// TIA Portal V17 export
// export: Created 2025-06-26T06:49:11.8212921Z, ExportSetting WithDefaults, DisplayName Totally Integrated Automation Portal, DisplayVersion V17 Update 8, DisplayName TIA Portal Openness, DisplayVersion V17 Update 8, DisplayName TIA Portal Version Control Interface, DisplayVersion V17, DisplayName STEP 7 Professional, DisplayVersion V17 Update 8, DisplayName STEP 7 Safety, DisplayVersion V17 Update 6, DisplayName WinCC Advanced, DisplayVersion V17 Update 8
FUNCTION_BLOCK "Regulation"   // FB5, FBD
{ S7_Optimized_Access := 'TRUE' }
VERSION : 0.1
// stored: AutoNumber true, IsIECCheckEnabled true, IsRetainMemResEnabled false, MemoryReserve 10, SetENOAutomatically false, UDAEnableTagReadback false
   VAR
      ExpValveCurrentPressureLimitation : Bool;
      enEmergencyStop { ExternalAccessible := 'False'; ExternalVisible := 'False'; ExternalWritable := 'False'} : Bool;
      CPCPumpRequestFromCPC { ExternalAccessible := 'False'; ExternalVisible := 'False'; ExternalWritable := 'False'} : Bool;   // Crankcase Pressure Control wants to run CPC pump
      CPCPumpRequestFromPurge { ExternalAccessible := 'False'; ExternalVisible := 'False'; ExternalWritable := 'False'} : Bool;   // Do compressor manifold purge
      ExpValveCurrentPressureTarged : Real;
      PerformanceControl_PerformanceRate : Real;
      PerformanceControl { ExternalAccessible := 'False'; ExternalVisible := 'False'; ExternalWritable := 'False'; S7_SetPoint := 'True'} : "PerformanceControl";   // Compressor setpoint
      SuperheatControl { ExternalAccessible := 'False'; ExternalVisible := 'False'; ExternalWritable := 'False'; S7_SetPoint := 'True'} : "SuperheatControl";   // Superheat setpoint
      PinchControl { ExternalAccessible := 'False'; ExternalVisible := 'False'; ExternalWritable := 'False'; S7_SetPoint := 'True'} : "PinchControl";
      CrankcaseOilHeating { ExternalAccessible := 'False'; ExternalVisible := 'False'; ExternalWritable := 'False'; S7_SetPoint := 'True'} : "OilHeating";
      MotorSpeedControl { ExternalAccessible := 'False'; ExternalVisible := 'False'; ExternalWritable := 'False'; S7_SetPoint := 'True'} : "MotorControl";
      SafetyRelay { ExternalAccessible := 'False'; ExternalVisible := 'False'; ExternalWritable := 'False'; S7_SetPoint := 'True'} : "fbSafetyRelay";
      CabinetTemperature { ExternalAccessible := 'False'; ExternalVisible := 'False'; ExternalWritable := 'False'; S7_SetPoint := 'True'} : "fbTemperatureController2";
      ContainerVentilation { ExternalAccessible := 'False'; ExternalVisible := 'False'; ExternalWritable := 'False'; S7_SetPoint := 'True'} : "fbPI_Regulator";
      CrankcasePressureControl { ExternalAccessible := 'False'; ExternalVisible := 'False'; ExternalWritable := 'False'; S7_SetPoint := 'True'} : "CrankcasePressureControl";
      OilSeparator { ExternalAccessible := 'False'; ExternalVisible := 'False'; ExternalWritable := 'False'; S7_SetPoint := 'True'} : "OilSeparator";
      ShaftSealCartridge { ExternalAccessible := 'False'; ExternalVisible := 'False'; ExternalWritable := 'False'; S7_SetPoint := 'True'} : "ShaftSealCartridge";
      LubricationPriming { ExternalAccessible := 'False'; ExternalVisible := 'False'; ExternalWritable := 'False'; S7_SetPoint := 'True'} : "LubricationPriming";
      ValveControl { ExternalAccessible := 'False'; ExternalVisible := 'False'; ExternalWritable := 'False'; S7_SetPoint := 'True'} : "ValveControl";
      PurgeControl { ExternalAccessible := 'False'; ExternalVisible := 'False'; ExternalWritable := 'False'; S7_SetPoint := 'True'} : "fbPurgeControl";
      FilterDryer { S7_SetPoint := 'True'} : "fbFilterDryer";
      OilRecovery { S7_SetPoint := 'True'} : "fbOilRecovery";
      RecuperatorBypass { S7_SetPoint := 'True'} : "fbNullRegulator";
      HeatSourceCycle { S7_SetPoint := 'True'} : "fbTrackingRegulator";
      HeatSourceCyclePIP { S7_SetPoint := 'True'} : "fbPIP_Regulator";
      HeatboosterSetpointPrev { ExternalAccessible := 'False'; ExternalVisible := 'False'; ExternalWritable := 'False'} : Real;   // TEST
      HeatSinkSetpointPrev { ExternalAccessible := 'False'; ExternalVisible := 'False'; ExternalWritable := 'False'} : Real;   // TEST
      HeatSourceSetpointPrev { ExternalAccessible := 'False'; ExternalVisible := 'False'; ExternalWritable := 'False'} : Real;   // TEST
      VariableSetpointPrev { ExternalAccessible := 'False'; ExternalVisible := 'False'; ExternalWritable := 'False'} : Real;
      RegulationTarget { ExternalAccessible := 'False'; ExternalVisible := 'False'; ExternalWritable := 'False'} : Int;   // TEST
      epHeatSinkControlActive { ExternalAccessible := 'False'; ExternalVisible := 'False'; ExternalWritable := 'False'} : Bool;
      epHeatSourceControlActive { ExternalAccessible := 'False'; ExternalVisible := 'False'; ExternalWritable := 'False'} : Bool;
      epVariableControlActive { ExternalAccessible := 'False'; ExternalVisible := 'False'; ExternalWritable := 'False'} : Bool;
      TEST1 : Bool;
   END_VAR
   VAR_TEMP
      AdditionalSuperHeat : Real;
      PerformanceSetpoint : Real;
      AdditionalSuperheatPinch : Real;
   END_VAR
   VAR_TEMP   // added for the SCL form of the ladder/FBD networks
      _w1 : Bool;
   END_VAR
BEGIN

REGION Network 1: Performance control
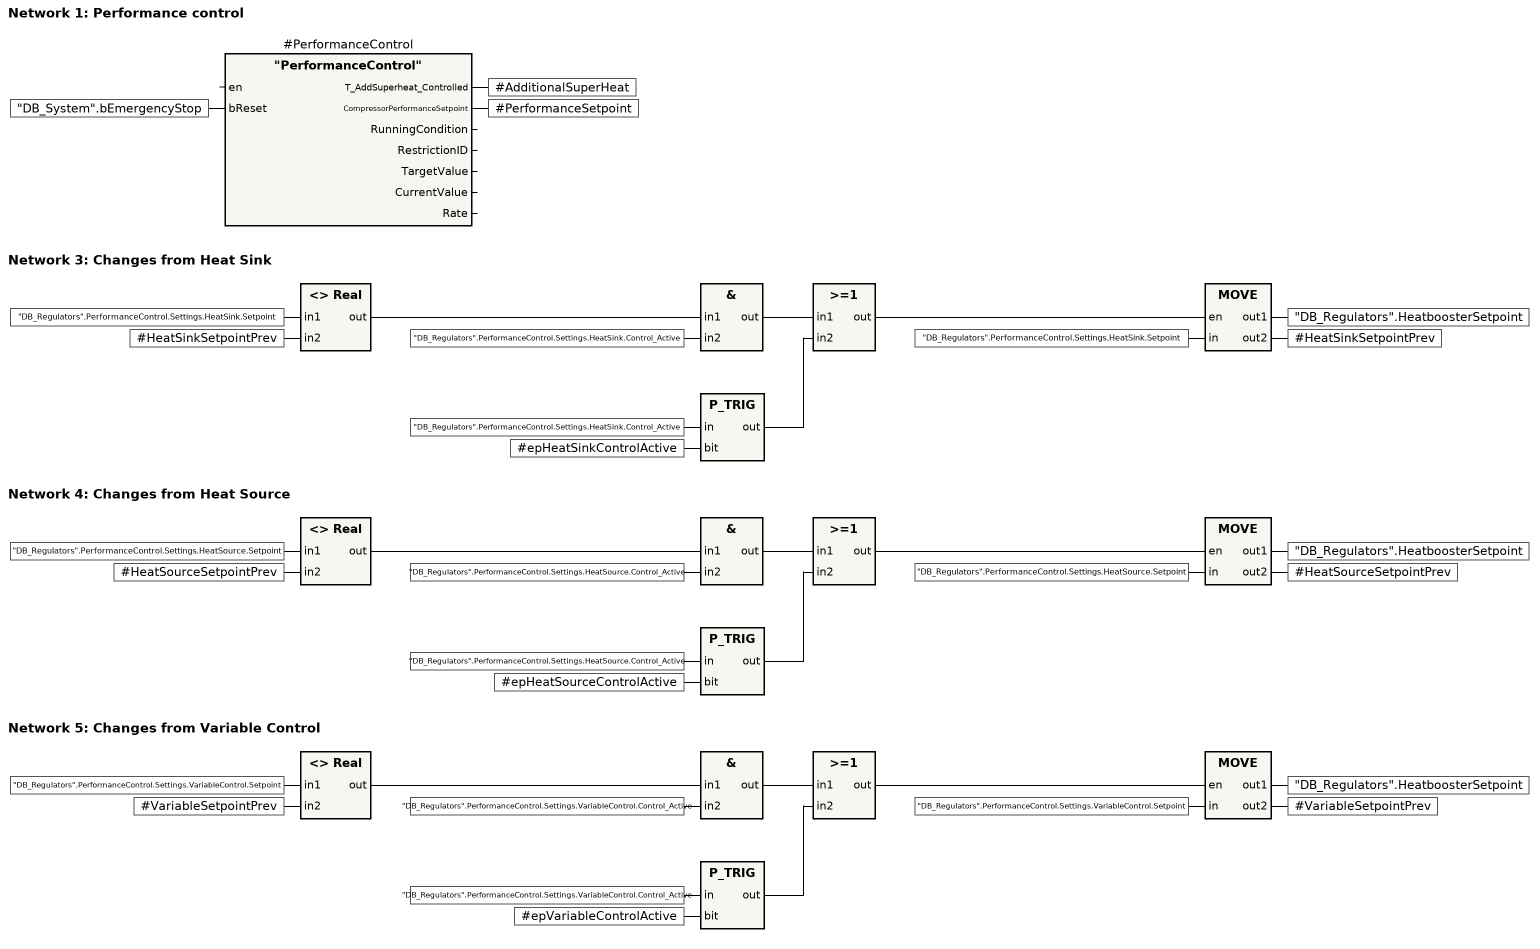
   #PerformanceControl(bReset := "DB_System".bEmergencyStop,   // "PerformanceControl"
                       T_AddSuperheat_Controlled => #AdditionalSuperHeat,
                       CompressorPerformanceSetpoint => #PerformanceSetpoint);
END_REGION

REGION Network 2 (SCL): Performance rate
   // Used in HMI only
   IF "DB_State".State."5_Warmup" OR "DB_State".State."6_Running" AND #PerformanceControl.RunningCondition = TRUE THEN
       #PerformanceControl_PerformanceRate := #MotorSpeedControl.NEngineSetpoint / 15 - #AdditionalSuperHeat / 50 * 30;
   ELSE
       #PerformanceControl_PerformanceRate := 0;
   END_IF;
END_REGION

REGION Network 3: Changes from Heat Sink
   // Propagate setpoint when controller is first activated, or if active and setpoint is changed
   #_w1 := "DB_Regulators".PerformanceControl.Settings.HeatSink.Control_Active AND NOT #epHeatSinkControlActive;   // rising edge
   #epHeatSinkControlActive := "DB_Regulators".PerformanceControl.Settings.HeatSink.Control_Active;
   IF (("DB_Regulators".PerformanceControl.Settings.HeatSink.Setpoint <> #HeatSinkSetpointPrev) AND "DB_Regulators".PerformanceControl.Settings.HeatSink.Control_Active) OR #_w1 THEN
       "DB_Regulators".HeatboosterSetpoint := "DB_Regulators".PerformanceControl.Settings.HeatSink.Setpoint;
       #HeatSinkSetpointPrev := "DB_Regulators".PerformanceControl.Settings.HeatSink.Setpoint;
   END_IF;
END_REGION

REGION Network 4: Changes from Heat Source
   // Propagate setpoint when controller is first activated, or if active and setpoint is changed
   #_w1 := "DB_Regulators".PerformanceControl.Settings.HeatSource.Control_Active AND NOT #epHeatSourceControlActive;   // rising edge
   #epHeatSourceControlActive := "DB_Regulators".PerformanceControl.Settings.HeatSource.Control_Active;
   IF (("DB_Regulators".PerformanceControl.Settings.HeatSource.Setpoint <> #HeatSourceSetpointPrev) AND "DB_Regulators".PerformanceControl.Settings.HeatSource.Control_Active) OR #_w1 THEN
       "DB_Regulators".HeatboosterSetpoint := "DB_Regulators".PerformanceControl.Settings.HeatSource.Setpoint;
       #HeatSourceSetpointPrev := "DB_Regulators".PerformanceControl.Settings.HeatSource.Setpoint;
   END_IF;
END_REGION

REGION Network 5: Changes from Variable Control
   // Propagate setpoint when controller is first activated, or if active and setpoint is changed
   #_w1 := "DB_Regulators".PerformanceControl.Settings.VariableControl.Control_Active AND NOT #epVariableControlActive;   // rising edge
   #epVariableControlActive := "DB_Regulators".PerformanceControl.Settings.VariableControl.Control_Active;
   IF (("DB_Regulators".PerformanceControl.Settings.VariableControl.Setpoint <> #VariableSetpointPrev) AND "DB_Regulators".PerformanceControl.Settings.VariableControl.Control_Active) OR #_w1 THEN
       "DB_Regulators".HeatboosterSetpoint := "DB_Regulators".PerformanceControl.Settings.VariableControl.Setpoint;
       #VariableSetpointPrev := "DB_Regulators".PerformanceControl.Settings.VariableControl.Setpoint;
   END_IF;
END_REGION

REGION Network 6 (SCL): Regulation target
   // No, I didn't suddenly develop a brain hemorrage, this mess here is on purpose:
   // 1. It is a sequence of separate IFs as it mirrors the logic in PerformanceControl
   // 2. It is tempting to re-use Restriction ID, but this can take on values other than the ones here, which we want to avoid. So the value has to be reconstructed.
   // Figure out which target is active
   "DB_Regulators".RegulationTarget := 0;  // in case none of the regulators are active, none of the IFs fire...
   IF "DB_Regulators".PerformanceControl.Settings.HeatSink.Control_Active THEN
       IF "DB_Regulators".PerformanceControl.Settings.HeatSink.UseFeedFlow THEN
           "DB_Regulators".RegulationTarget := 2;
       ELSE
           "DB_Regulators".RegulationTarget := 1;
       END_IF;
   END_IF;

   IF "DB_Regulators".PerformanceControl.Settings.HeatSource.Control_Active THEN
       IF "DB_Regulators".PerformanceControl.Settings.HeatSource.UseFeedFlow THEN
           "DB_Regulators".RegulationTarget := 4;
       ELSE
           "DB_Regulators".RegulationTarget := 3;
       END_IF;
   END_IF;

   IF "DB_Regulators".PerformanceControl.Settings.VariableControl.Control_Active AND "DB_Regulators".PerformanceControl.Settings.VariableControl.ReferenceID > 0 THEN
       "DB_Regulators".RegulationTarget := 6;
   END_IF;
END_REGION

REGION Network 7: Changes from DB_Regulators
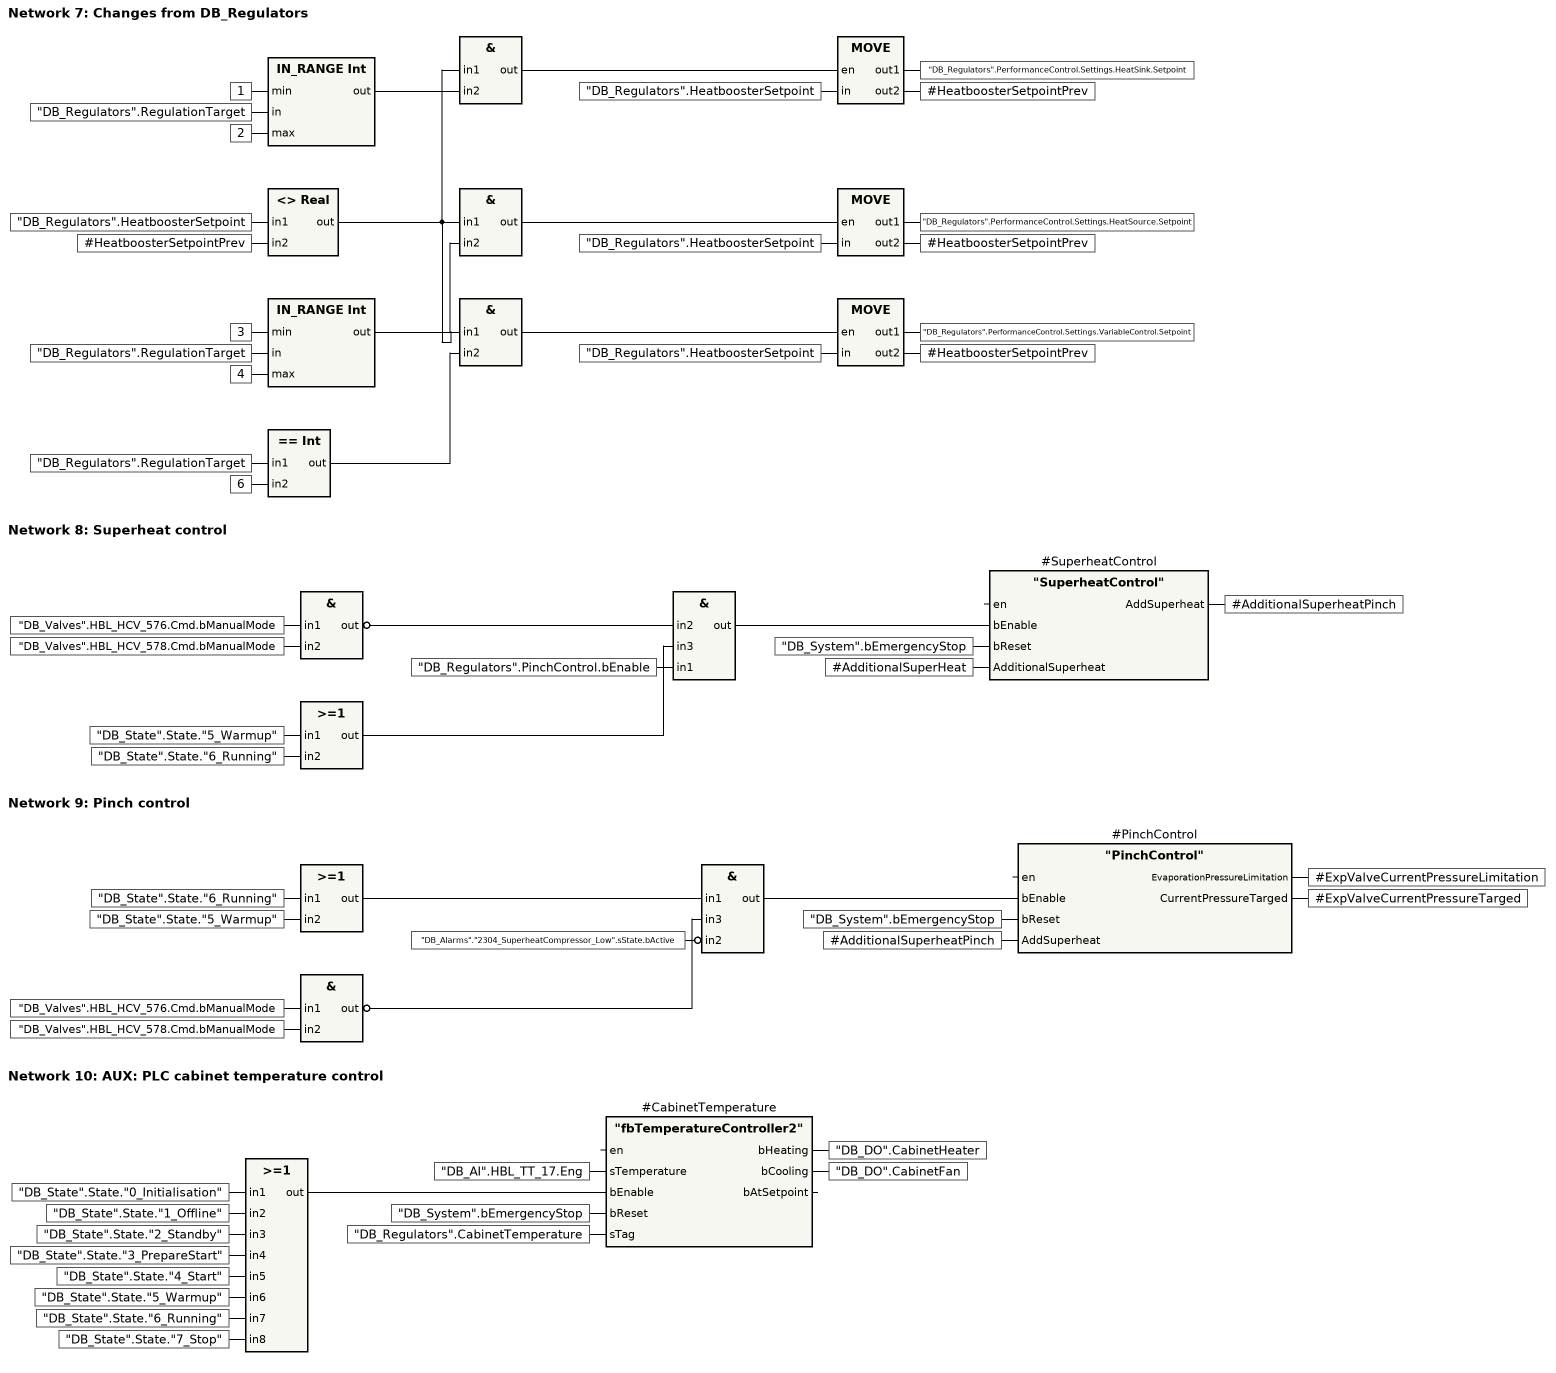
   #_w1 := "DB_Regulators".HeatboosterSetpoint <> #HeatboosterSetpointPrev;
   IF #_w1 AND (1 <= "DB_Regulators".RegulationTarget) AND ("DB_Regulators".RegulationTarget <= 2) THEN
       "DB_Regulators".PerformanceControl.Settings.HeatSink.Setpoint := "DB_Regulators".HeatboosterSetpoint;
       #HeatboosterSetpointPrev := "DB_Regulators".HeatboosterSetpoint;
   END_IF;
   IF #_w1 AND (3 <= "DB_Regulators".RegulationTarget) AND ("DB_Regulators".RegulationTarget <= 4) THEN
       "DB_Regulators".PerformanceControl.Settings.HeatSource.Setpoint := "DB_Regulators".HeatboosterSetpoint;
       #HeatboosterSetpointPrev := "DB_Regulators".HeatboosterSetpoint;
   END_IF;
   IF #_w1 AND ("DB_Regulators".RegulationTarget = 6) THEN
       "DB_Regulators".PerformanceControl.Settings.VariableControl.Setpoint := "DB_Regulators".HeatboosterSetpoint;
       #HeatboosterSetpointPrev := "DB_Regulators".HeatboosterSetpoint;
   END_IF;
END_REGION

REGION Network 8: Superheat control
   #SuperheatControl(bEnable := NOT ("DB_Valves".HBL_HCV_576.Cmd.bManualMode AND "DB_Valves".HBL_HCV_578.Cmd.bManualMode) AND ("DB_State".State."5_Warmup" OR "DB_State".State."6_Running") AND "DB_Regulators".PinchControl.bEnable,   // "SuperheatControl"
                     bReset := "DB_System".bEmergencyStop,
                     AdditionalSuperheat := #AdditionalSuperHeat,
                     AddSuperheat => #AdditionalSuperheatPinch);
END_REGION

REGION Network 9: Pinch control
   #PinchControl(bEnable := ("DB_State".State."6_Running" OR "DB_State".State."5_Warmup") AND NOT ("DB_Valves".HBL_HCV_576.Cmd.bManualMode AND "DB_Valves".HBL_HCV_578.Cmd.bManualMode) AND NOT "DB_Alarms"."2304_SuperheatCompressor_Low".sState.bActive,   // "PinchControl"
                 bReset := "DB_System".bEmergencyStop,
                 AddSuperheat := #AdditionalSuperheatPinch,
                 EvaporationPressureLimitation => #ExpValveCurrentPressureLimitation,
                 CurrentPressureTarged => #ExpValveCurrentPressureTarged);
END_REGION

REGION Network 10: AUX: PLC cabinet temperature control
   // Runs all the time, as the cabinet is running all the time...
   #CabinetTemperature(sTemperature := "DB_AI".HBL_TT_17.Eng,   // "fbTemperatureController2"
                       bEnable := "DB_State".State."0_Initialisation" OR "DB_State".State."1_Offline" OR "DB_State".State."2_Standby" OR "DB_State".State."3_PrepareStart" OR "DB_State".State."4_Start" OR "DB_State".State."5_Warmup" OR "DB_State".State."6_Running" OR "DB_State".State."7_Stop",
                       bReset := "DB_System".bEmergencyStop,
                       sTag := "DB_Regulators".CabinetTemperature,
                       bHeating => "DB_DO".CabinetHeater,
                       bCooling => "DB_DO".CabinetFan);
END_REGION

REGION Network 11: AUX: Crankcase oil heater control
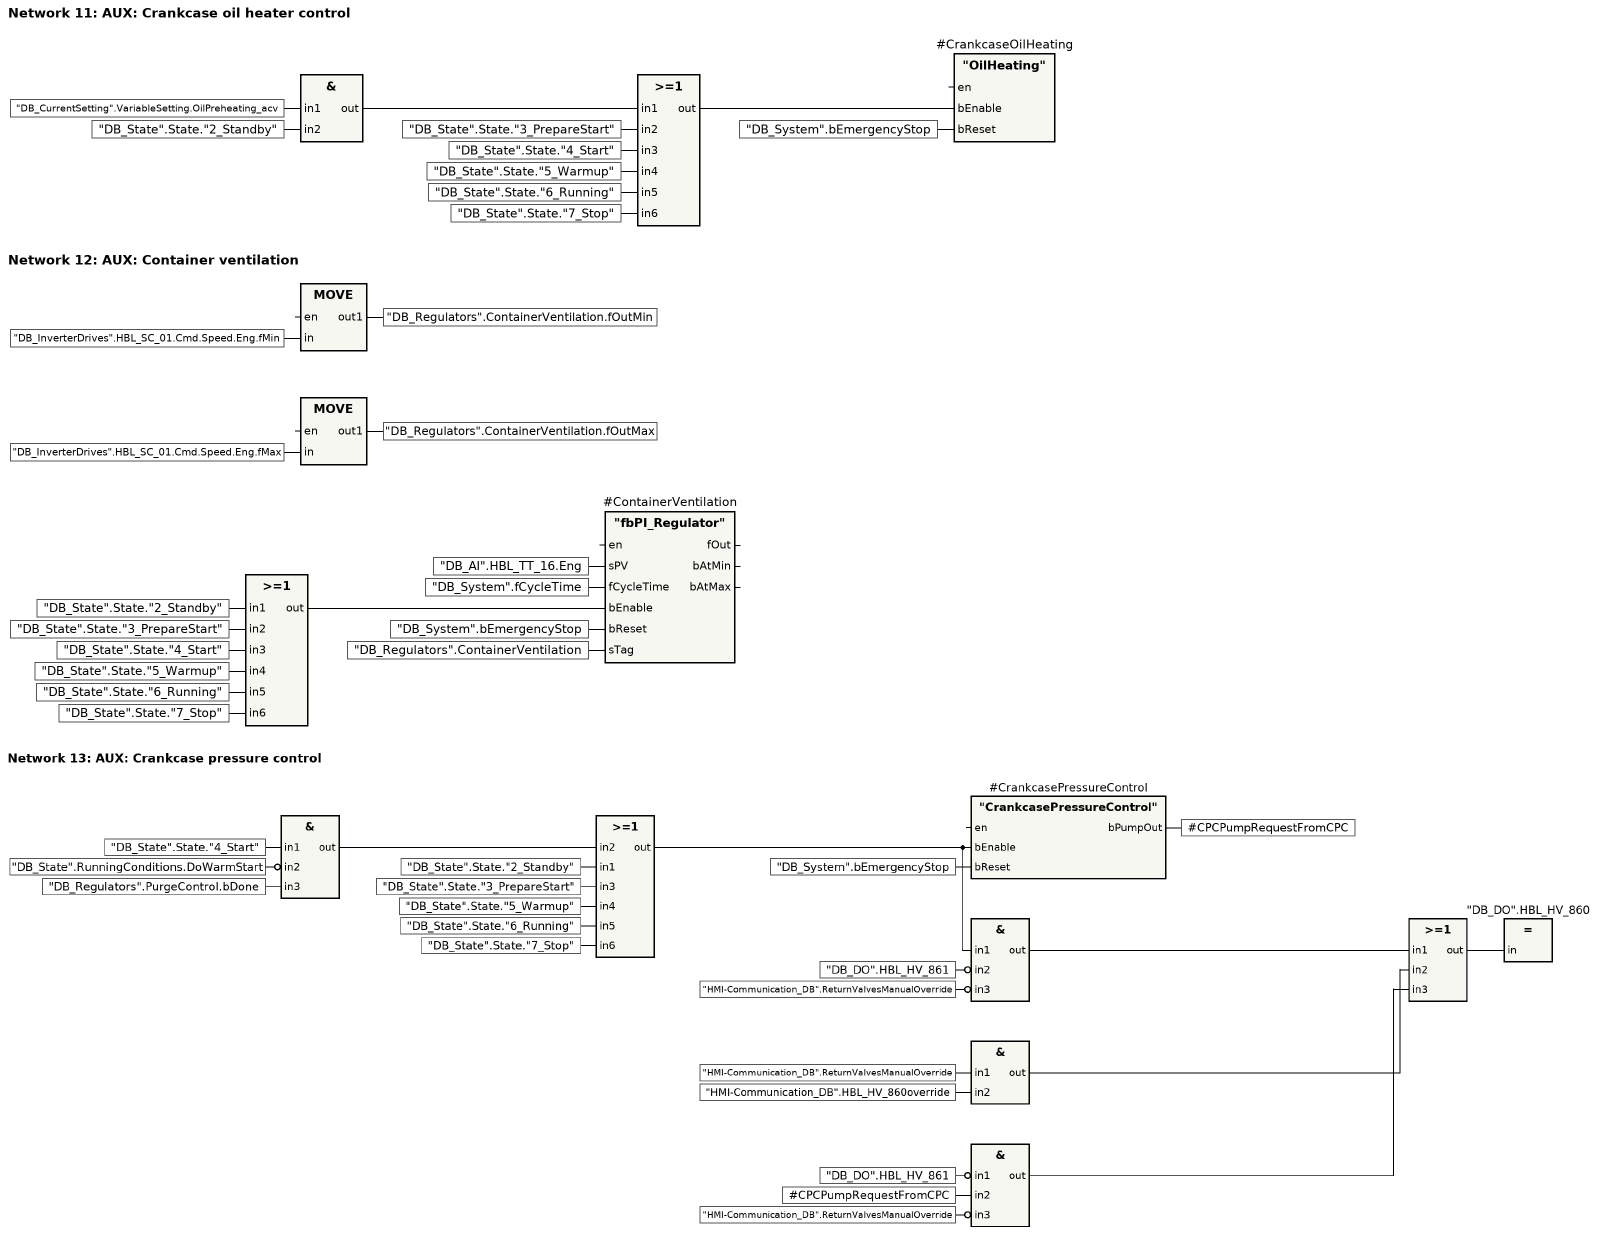
   #CrankcaseOilHeating(bEnable := ("DB_CurrentSetting".VariableSetting.OilPreheating_acv AND "DB_State".State."2_Standby") OR "DB_State".State."3_PrepareStart" OR "DB_State".State."4_Start" OR "DB_State".State."5_Warmup" OR "DB_State".State."6_Running" OR "DB_State".State."7_Stop",   // "OilHeating"
                        bReset := "DB_System".bEmergencyStop);
END_REGION

REGION Network 12: AUX: Container ventilation
   // Manually copy the actuator min & max to the regulator min & max. This is not automatically true for all regulators
   // ##FIX: Hack the start signal, ugliness alert
   "DB_Regulators".ContainerVentilation.fOutMin := "DB_InverterDrives".HBL_SC_01.Cmd.Speed.Eng.fMin;
   "DB_Regulators".ContainerVentilation.fOutMax := "DB_InverterDrives".HBL_SC_01.Cmd.Speed.Eng.fMax;
   #ContainerVentilation(sPV := "DB_AI".HBL_TT_16.Eng,   // "fbPI_Regulator"
                         fCycleTime := "DB_System".fCycleTime,
                         bEnable := "DB_State".State."2_Standby" OR "DB_State".State."3_PrepareStart" OR "DB_State".State."4_Start" OR "DB_State".State."5_Warmup" OR "DB_State".State."6_Running" OR "DB_State".State."7_Stop",
                         bReset := "DB_System".bEmergencyStop,
                         sTag := "DB_Regulators".ContainerVentilation);
END_REGION

REGION Network 13: AUX: Crankcase pressure control
   // Disable the controller temporarily in State 4 Start when doing a cold start
   #_w1 := ("DB_State".State."4_Start" AND NOT "DB_State".RunningConditions.DoWarmStart AND "DB_Regulators".PurgeControl.bDone) OR "DB_State".State."2_Standby" OR "DB_State".State."3_PrepareStart" OR "DB_State".State."5_Warmup" OR "DB_State".State."6_Running" OR "DB_State".State."7_Stop";
   #CrankcasePressureControl(bEnable := #_w1,   // "CrankcasePressureControl"
                           bReset := "DB_System".bEmergencyStop,
                           bPumpOut => #CPCPumpRequestFromCPC);
   "DB_DO".HBL_HV_860 := (#_w1 AND NOT "DB_DO".HBL_HV_861 AND NOT "HMI-Communication_DB".ReturnValvesManualOverride) OR ("HMI-Communication_DB".ReturnValvesManualOverride AND "HMI-Communication_DB".HBL_HV_860override) OR (NOT "DB_DO".HBL_HV_861 AND #CPCPumpRequestFromCPC AND NOT "HMI-Communication_DB".ReturnValvesManualOverride);
END_REGION

REGION Network 14: AUX: Oil separator level control
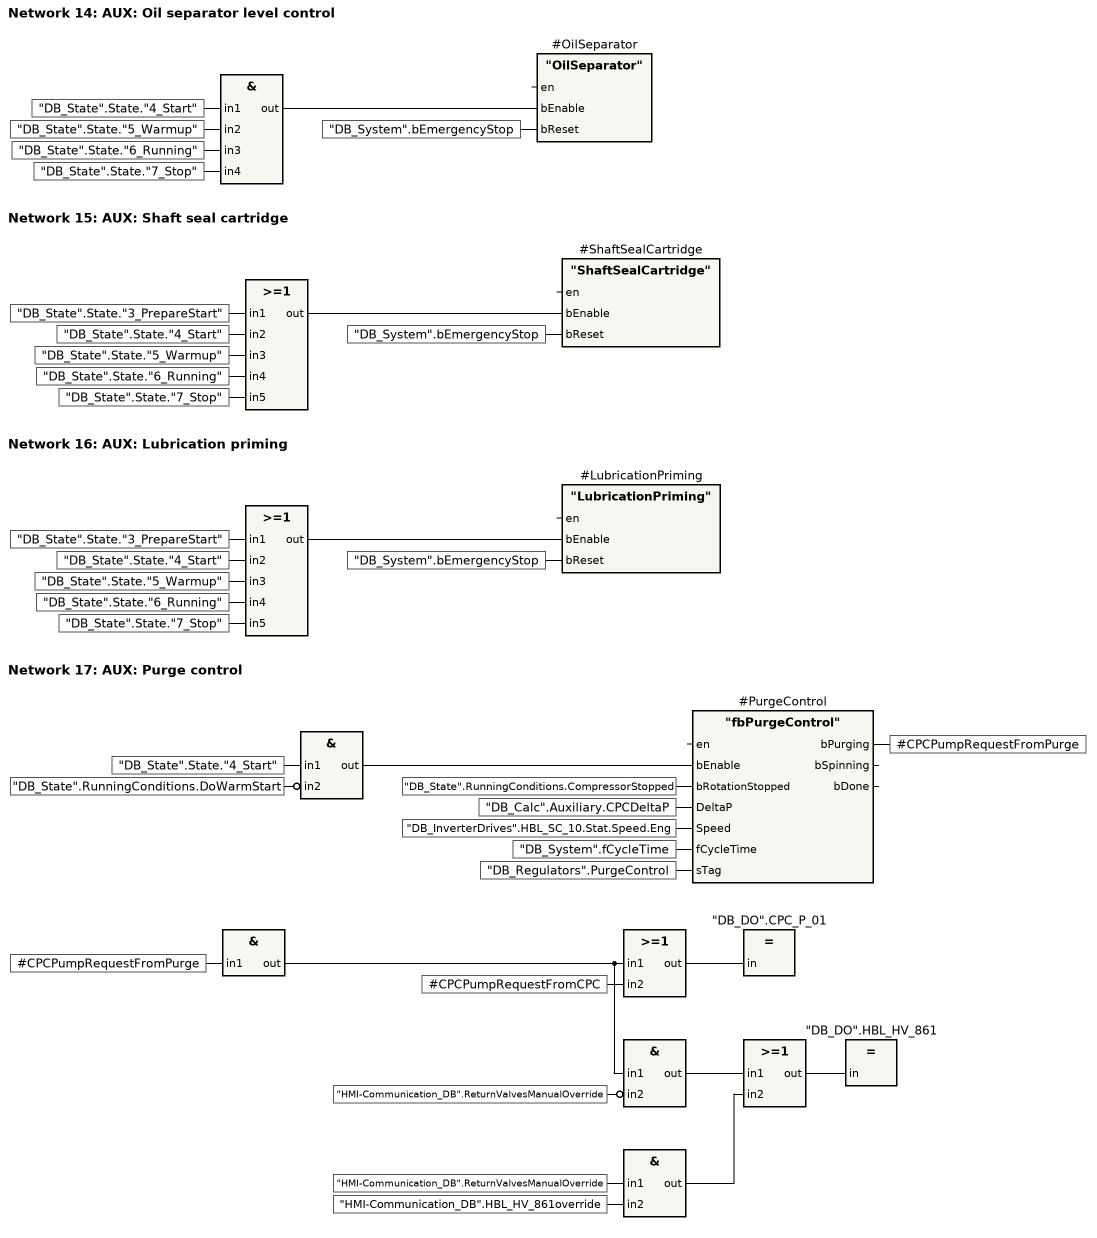
   #OilSeparator(bEnable := "DB_State".State."4_Start" AND "DB_State".State."5_Warmup" AND "DB_State".State."6_Running" AND "DB_State".State."7_Stop",   // "OilSeparator"
                 bReset := "DB_System".bEmergencyStop);
END_REGION

REGION Network 15: AUX: Shaft seal cartridge
   #ShaftSealCartridge(bEnable := "DB_State".State."3_PrepareStart" OR "DB_State".State."4_Start" OR "DB_State".State."5_Warmup" OR "DB_State".State."6_Running" OR "DB_State".State."7_Stop",   // "ShaftSealCartridge"
                       bReset := "DB_System".bEmergencyStop);
END_REGION

REGION Network 16: AUX: Lubrication priming
   #LubricationPriming(bEnable := "DB_State".State."3_PrepareStart" OR "DB_State".State."4_Start" OR "DB_State".State."5_Warmup" OR "DB_State".State."6_Running" OR "DB_State".State."7_Stop",   // "LubricationPriming"
                       bReset := "DB_System".bEmergencyStop);
END_REGION

REGION Network 17: AUX: Purge control
   // Note: HBL-XV-05 takes priority over HBL-XV-04
   #PurgeControl(bEnable := "DB_State".State."4_Start" AND NOT "DB_State".RunningConditions.DoWarmStart,   // "fbPurgeControl"
                 bRotationStopped := "DB_State".RunningConditions.CompressorStopped,
                 DeltaP := "DB_Calc".Auxiliary.CPCDeltaP,
                 Speed := "DB_InverterDrives".HBL_SC_10.Stat.Speed.Eng,
                 fCycleTime := "DB_System".fCycleTime,
                 sTag := "DB_Regulators".PurgeControl,
                 bPurging => #CPCPumpRequestFromPurge);
   "DB_DO".CPC_P_01 := #CPCPumpRequestFromPurge OR #CPCPumpRequestFromCPC;
   "DB_DO".HBL_HV_861 := (#CPCPumpRequestFromPurge AND NOT "HMI-Communication_DB".ReturnValvesManualOverride) OR ("HMI-Communication_DB".ReturnValvesManualOverride AND "HMI-Communication_DB".HBL_HV_861override);
END_REGION

REGION Network 18: AUX: Compressor manifold oil return
   // This is still up in the air what this will be
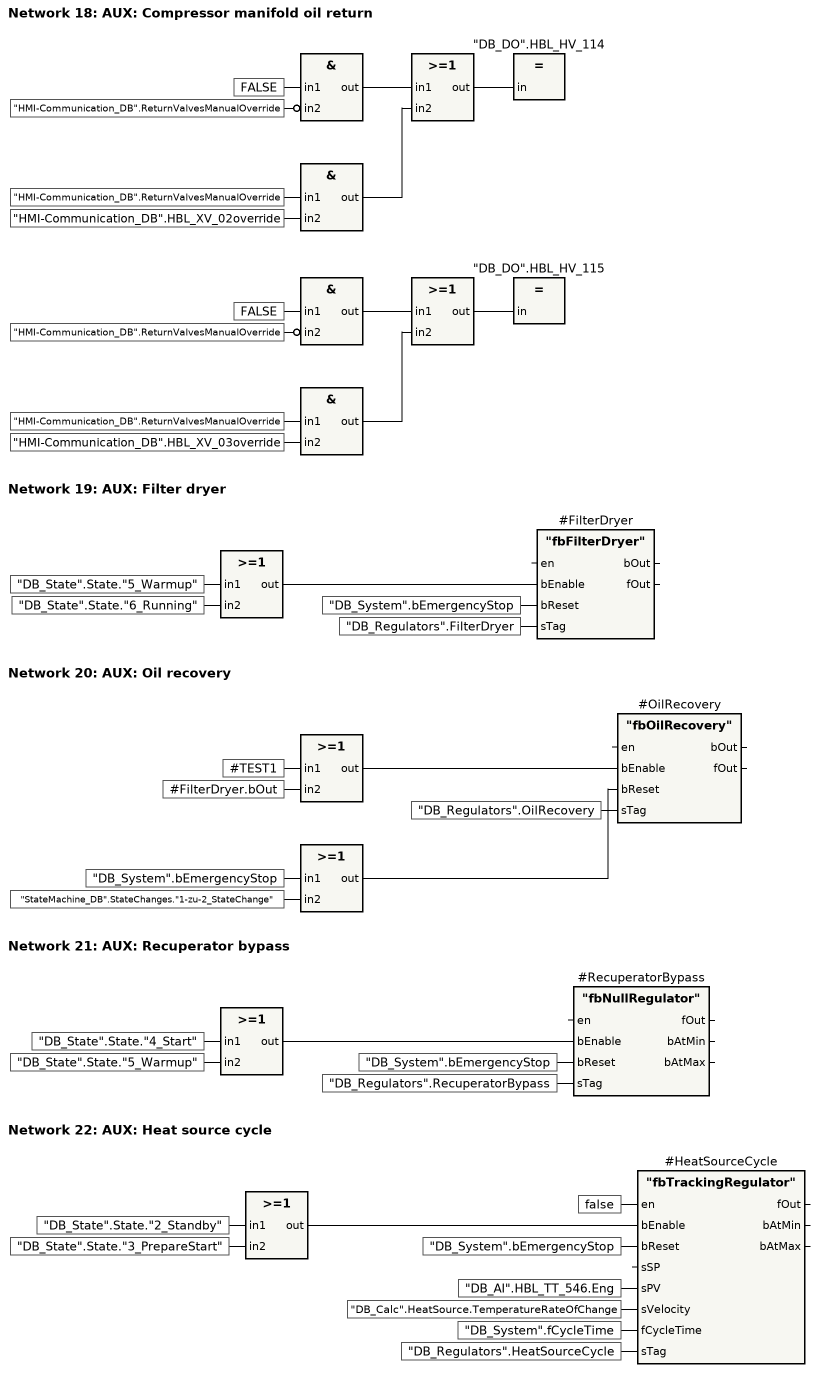
   "DB_DO".HBL_HV_114 := (FALSE AND NOT "HMI-Communication_DB".ReturnValvesManualOverride) OR ("HMI-Communication_DB".ReturnValvesManualOverride AND "HMI-Communication_DB".HBL_XV_02override);
   "DB_DO".HBL_HV_115 := (FALSE AND NOT "HMI-Communication_DB".ReturnValvesManualOverride) OR ("HMI-Communication_DB".ReturnValvesManualOverride AND "HMI-Communication_DB".HBL_XV_03override);
END_REGION

REGION Network 19: AUX: Filter dryer
   #FilterDryer(bEnable := "DB_State".State."5_Warmup" OR "DB_State".State."6_Running",   // "fbFilterDryer"
                bReset := "DB_System".bEmergencyStop,
                sTag := "DB_Regulators".FilterDryer);
END_REGION

REGION Network 20: AUX: Oil recovery
   // Run only when filter dryer is also running
   #OilRecovery(bEnable := #TEST1 OR #FilterDryer.bOut,   // "fbOilRecovery"
                bReset := "DB_System".bEmergencyStop OR "StateMachine_DB".StateChanges."1-zu-2_StateChange",
                sTag := "DB_Regulators".OilRecovery);
END_REGION

REGION Network 21: AUX: Recuperator bypass
   #RecuperatorBypass(bEnable := "DB_State".State."4_Start" OR "DB_State".State."5_Warmup",   // "fbNullRegulator"
                      bReset := "DB_System".bEmergencyStop,
                      sTag := "DB_Regulators".RecuperatorBypass);
END_REGION

REGION Network 22: AUX: Heat source cycle
   IF false THEN
       #HeatSourceCycle(bEnable := "DB_State".State."2_Standby" OR "DB_State".State."3_PrepareStart",   // "fbTrackingRegulator"
                        bReset := "DB_System".bEmergencyStop,
                        sPV := "DB_AI".HBL_TT_546.Eng,
                        sVelocity := "DB_Calc".HeatSource.TemperatureRateOfChange,
                        fCycleTime := "DB_System".fCycleTime,
                        sTag := "DB_Regulators".HeatSourceCycle);
   END_IF;
END_REGION

REGION Network 23: AUX: Heat source cycle PIP
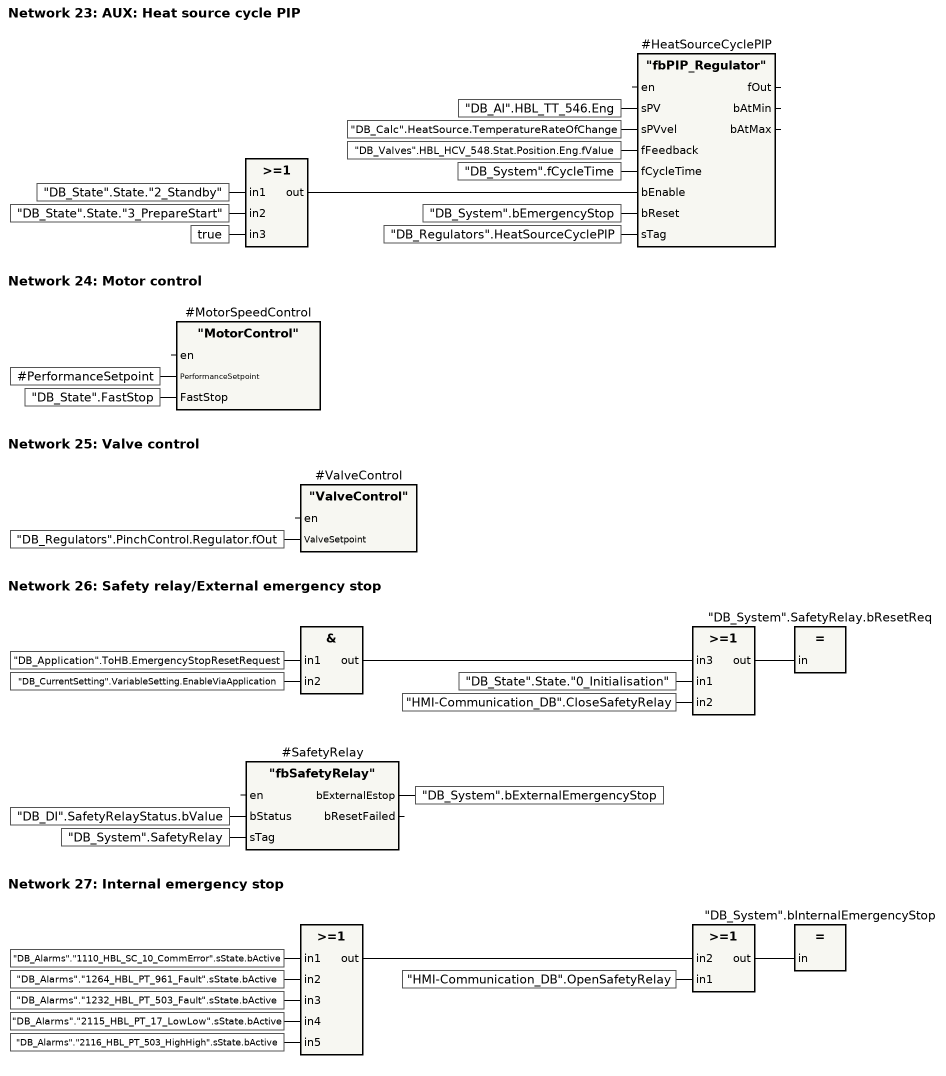
   #HeatSourceCyclePIP(sPV := "DB_AI".HBL_TT_546.Eng,   // "fbPIP_Regulator"
                       sPVvel := "DB_Calc".HeatSource.TemperatureRateOfChange,
                       fFeedback := "DB_Valves".HBL_HCV_548.Stat.Position.Eng.fValue,
                       fCycleTime := "DB_System".fCycleTime,
                       bEnable := "DB_State".State."2_Standby" OR "DB_State".State."3_PrepareStart" OR true,
                       bReset := "DB_System".bEmergencyStop,
                       sTag := "DB_Regulators".HeatSourceCyclePIP);
END_REGION

REGION Network 24: Motor control
   // Note this has to come after all regulators which set the motor speed
   #MotorSpeedControl(PerformanceSetpoint := #PerformanceSetpoint, FastStop := "DB_State".FastStop);   // "MotorControl"
END_REGION

REGION Network 25: Valve control
   #ValveControl(ValveSetpoint := "DB_Regulators".PinchControl.Regulator.fOut);   // "ValveControl"
END_REGION

REGION Network 26: Safety relay/External emergency stop
   "DB_System".SafetyRelay.bResetReq := ("DB_Application".ToHB.EmergencyStopResetRequest AND "DB_CurrentSetting".VariableSetting.EnableViaApplication) OR "DB_State".State."0_Initialisation" OR "HMI-Communication_DB".CloseSafetyRelay;
   #SafetyRelay(bStatus := "DB_DI".SafetyRelayStatus.bValue,   // "fbSafetyRelay"
                sTag := "DB_System".SafetyRelay,
                bExternalEstop => "DB_System".bExternalEmergencyStop);
END_REGION

REGION Network 27: Internal emergency stop
   // The alarms in this list should also be in the Critical alarms list in FB32 AlarmManagement.
   // HBL-PT-17 : lubrication failure, stop compressor (or fault in this sensor)
   // HBL-PT-503: compressor discharge overpressure, stop the compressor (or fault in this sensor)
   // HBL-SC-10: compressor inverter communication loss, no other way to shut it down except by hardwired emergency stop.
   "DB_System".bInternalEmergencyStop := "DB_Alarms"."1110_HBL_SC_10_CommError".sState.bActive OR "DB_Alarms"."1264_HBL_PT_961_Fault".sState.bActive OR "DB_Alarms"."1232_HBL_PT_503_Fault".sState.bActive OR "DB_Alarms"."2115_HBL_PT_17_LowLow".sState.bActive OR "DB_Alarms"."2116_HBL_PT_503_HighHigh".sState.bActive OR "HMI-Communication_DB".OpenSafetyRelay;
END_REGION

REGION Network 28: Emergency stop
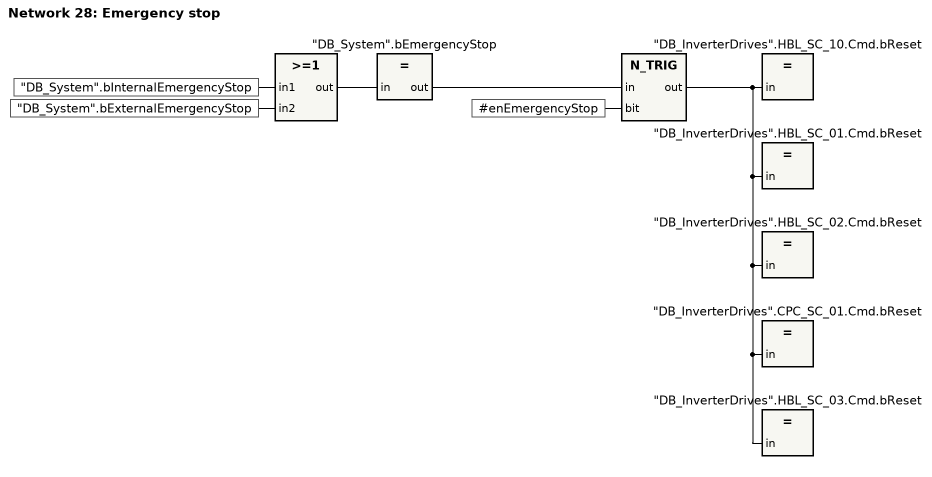
   "DB_System".bEmergencyStop := "DB_System".bInternalEmergencyStop OR "DB_System".bExternalEmergencyStop;
   #_w1 := NOT "DB_System".bEmergencyStop AND #enEmergencyStop;   // falling edge
   #enEmergencyStop := "DB_System".bEmergencyStop;
   "DB_InverterDrives".HBL_SC_10.Cmd.bReset := #_w1;
   "DB_InverterDrives".HBL_SC_01.Cmd.bReset := #_w1;
   "DB_InverterDrives".HBL_SC_02.Cmd.bReset := #_w1;
   "DB_InverterDrives".CPC_SC_01.Cmd.bReset := #_w1;
   "DB_InverterDrives".HBL_SC_03.Cmd.bReset := #_w1;
END_REGION

REGION Network 29: Manual mode warning
   // One or more regulators or actuators is in manual mode.
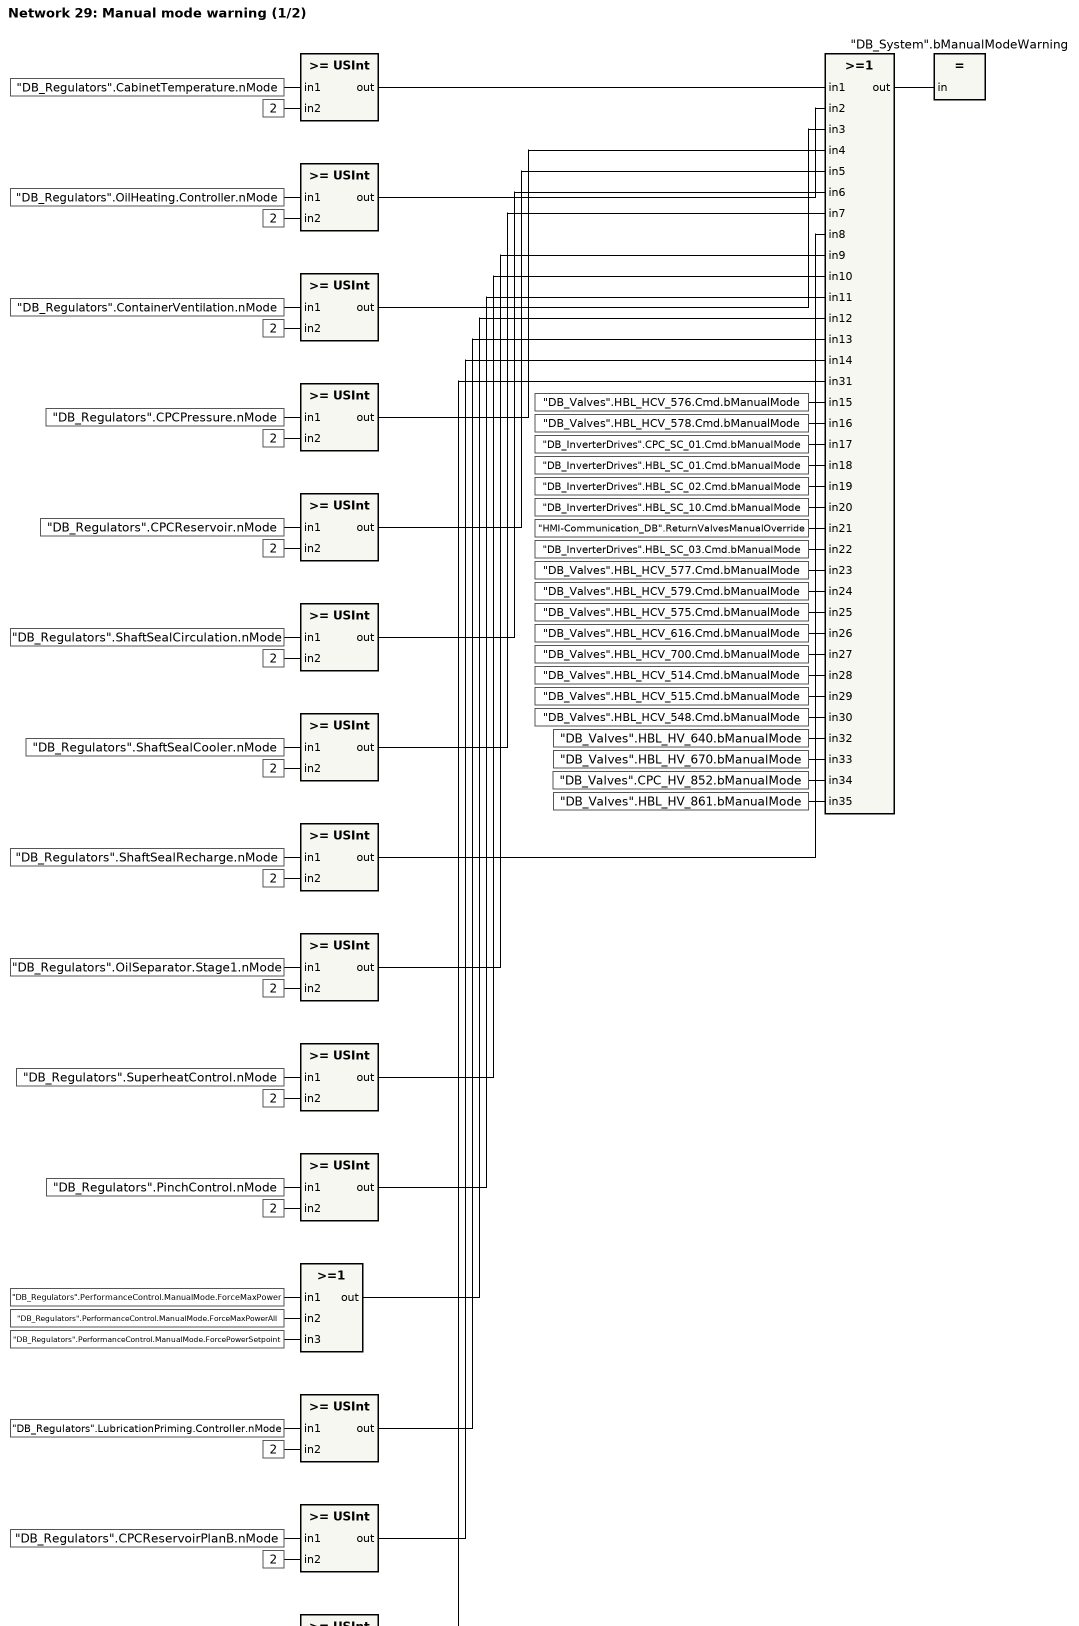
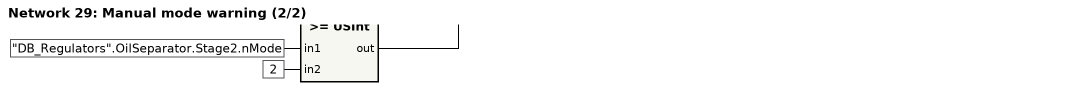
   "DB_System".bManualModeWarning := ("DB_Regulators".CabinetTemperature.nMode >= 2) OR ("DB_Regulators".OilHeating.Controller.nMode >= 2) OR ("DB_Regulators".ContainerVentilation.nMode >= 2) OR ("DB_Regulators".CPCPressure.nMode >= 2) OR ("DB_Regulators".CPCReservoir.nMode >= 2) OR ("DB_Regulators".ShaftSealCirculation.nMode >= 2) OR ("DB_Regulators".ShaftSealCooler.nMode >= 2) OR ("DB_Regulators".ShaftSealRecharge.nMode >= 2) OR ("DB_Regulators".OilSeparator.Stage1.nMode >= 2) OR ("DB_Regulators".SuperheatControl.nMode >= 2) OR ("DB_Regulators".PinchControl.nMode >= 2) OR "DB_Regulators".PerformanceControl.ManualMode.ForceMaxPower OR "DB_Regulators".PerformanceControl.ManualMode.ForceMaxPowerAll OR "DB_Regulators".PerformanceControl.ManualMode.ForcePowerSetpoint OR ("DB_Regulators".LubricationPriming.Controller.nMode >= 2) OR ("DB_Regulators".CPCReservoirPlanB.nMode >= 2) OR ("DB_Regulators".OilSeparator.Stage2.nMode >= 2) OR "DB_Valves".HBL_HCV_576.Cmd.bManualMode OR "DB_Valves".HBL_HCV_578.Cmd.bManualMode OR "DB_InverterDrives".CPC_SC_01.Cmd.bManualMode OR "DB_InverterDrives".HBL_SC_01.Cmd.bManualMode OR "DB_InverterDrives".HBL_SC_02.Cmd.bManualMode OR "DB_InverterDrives".HBL_SC_10.Cmd.bManualMode OR "HMI-Communication_DB".ReturnValvesManualOverride OR "DB_InverterDrives".HBL_SC_03.Cmd.bManualMode OR "DB_Valves".HBL_HCV_577.Cmd.bManualMode OR "DB_Valves".HBL_HCV_579.Cmd.bManualMode OR "DB_Valves".HBL_HCV_575.Cmd.bManualMode OR "DB_Valves".HBL_HCV_616.Cmd.bManualMode OR "DB_Valves".HBL_HCV_700.Cmd.bManualMode OR "DB_Valves".HBL_HCV_514.Cmd.bManualMode OR "DB_Valves".HBL_HCV_515.Cmd.bManualMode OR "DB_Valves".HBL_HCV_548.Cmd.bManualMode OR "DB_Valves".HBL_HV_640.bManualMode OR "DB_Valves".HBL_HV_670.bManualMode OR "DB_Valves".CPC_HV_852.bManualMode OR "DB_Valves".HBL_HV_861.bManualMode;
END_REGION
END_FUNCTION_BLOCK
